// TIA Portal V20 export
TYPE "LER_typeThicknessTrackingData"
// stored: Access Published
   STRUCT
      resultDataThickness { ExternalWritable := 'False'} : Array[0..3] of Real;
      resultOK { ExternalWritable := 'False'} : Bool;
      resultNG { ExternalWritable := 'False'} : Bool;
      complete { ExternalWritable := 'False'} : Bool;
   END_STRUCT;
END_TYPE
